// TIA Portal V16 export
// export: Created 2021-11-12T13:33:45.7137772Z, ExportSetting WithDefaults, DisplayName Totally Integrated Automation Portal, DisplayVersion V16 Update 3, DisplayName TIA Portal Version Control Interface, DisplayVersion V16 Update 2, DisplayName TIA Portal Openness, DisplayVersion V16 Update 3, DisplayName SINAMICS Startdrive Advanced, DisplayVersion V16 Update 5, DisplayName SINAMICS Startdrive G130, G150, S120, S150, SINAMICS MV, S210, DisplayVersion V16 Update 5, DisplayName SINAMICS Startdrive G110M, G120, G120C, G120D, G120P, G115D, DisplayVersion V16 Update 5, DisplayName STEP 7 Professional, DisplayVersion V16 Update 3, DisplayName STEP 7 Safety, DisplayVersion V16, DisplayName WinCC UA Professional, DisplayVersion V16 Update 3
DATA_BLOCK "Dummy_DB"   // DB66
{ S7_Optimized_Access := 'TRUE' }
VERSION : 0.1
// stored: AutoNumber false, DBAccessibleFromOPCUA true, IsOnlyStoredInLoadMemory false, IsRetainMemResEnabled false, IsWriteProtectedInAS false, MemoryReserve 100
   VAR
      R_STATUS_S : "UDT_RobotABB_Status_specific";
      R_GRIPPERSTATUS_S : "UDT_RobotGripper_Status_specific";
      R_STATUS_M : "UDT_Status_main";
      R_GRIPPERCOMMANDS : "UDT_RobotGripper_Command";
      R_PARAM : "UDT_RobotABB_Parameter";
      DSS : "UDT_DriveRobotABB_Status_specific";
      RSS : "UDT_RobotABB_Status_specific";
      R_COMMANDS : "UDT_RobotABB_Command";
      ZS : "UDT_Zone_Status_specific";
      R_DRIVESTATUS_S : "UDT_DriveRobotABB_Status_specific";
      SM : "UDT_Status_main";
      R_GRIPPERSTATUS : "UDT_Status_main";
      D2SS : "UDT_Drive2_Status_specific";
      D2C : "UDT_Drive2_Command";
      V2WBSS : "UDT_Valve2WB_Status_specific";
      V2WBC : "UDT_Valve2WB_Command";
      LiveBit { S7_SetPoint := 'True'} : Bool;
      TestNumber { S7_SetPoint := 'True'} : Int;
   END_VAR
BEGIN
END_DATA_BLOCK
